FUNCTION_BLOCK FB_StateMachine
VAR_INPUT
	bUltrasonicSensor: BOOL;
	bUpperLimitSwitch: BOOL;
	bLowerLimitSwitch: BOOL;
	bPhotocell: BOOL;
END_VAR
VAR_OUTPUT
	bMotorUp: BOOL;
	bMotorDown: BOOL;
END_VAR
VAR
	fBTon: TON;
	state : E_States;
END_VAR

CASE state OF
	E_States.eClosed:
		bMotorUp := FALSE;
		bMotorDown := FALSE;
		IF bUltrasonicSensor THEN
			state:= E_States.eOpening;
		END_IF
	
	E_States.eOpening:
		bMotorUp := TRUE;
		bMotorDown := FALSE;
		IF bUpperLimitSwitch THEN
			state:= E_States.eOpened;
		END_IF

	E_States.eOpened:
		fBTon(IN := NOT bPhotocell AND NOT bUltrasonicSensor , 
			  PT:=T#5S, 
			  Q=>,
			  ET=>);
		bMotorUp := FALSE;
		bMotorDown := FALSE;
		IF fBTon.Q THEN
			state:= E_States.eClosing;
		END_IF
	
	E_States.eClosing:
		fBTon(IN := FALSE);
		bMotorUp := FALSE;
		bMotorDown := TRUE;
		IF bPhotocell OR bUltrasonicSensor THEN
			state:= E_States.eOpening;
		ELSIF bLowerLimitSwitch THEN
			state:= E_States.eClosed;
		END_IF
END_CASE

END_FUNCTION_BLOCK

(* stored: Version 1.1.0.1, ProductVersion 3.1.4024.12
   POU FB_StateMachine: Id {e5816da5-9d48-4cc9-a5b5-8004a7c5ec6a}, SpecialFunc None *)
